(* 
| :Description: This function block represent basic TCP/IP client. 
| Use MR_Init to connect to the server. 
| To send data to server use MR_AppendToSendBuffer, use FUN_StringToTcpBufferData to convert string into structure of bytes.
| If the lenght of LastRecivedMessage is bigger than 0 then you recived message from server, use FUN_TcpBufferDataToString to copy it to string message.
| To close the connection use MR_Abort.
*)
FUNCTION_BLOCK FB_TcpClient EXTENDS FB_TcpDevice
VAR		
	(* Function blocks *)
	fbSocketConnect : FB_SocketConnect;		(* FB used to connect the client to remote server *)
END_VAR
(*
Version history:

+-------------+------------+----------------+----------+-------------------------------------------------------------------------------------+
|Date         | Version    | created under  | Author   | Remark                                                                              |
+=============+============+================+==========+=====================================================================================+
|2022-01      | 1.0.0.0    | V3.1.4024.22   | ADBO     | Function block created                                                              |
+-------------+------------+----------------+----------+-------------------------------------------------------------------------------------+
|2022-02      | 1.1.0.0    | V3.1.4024.22   | ADBO     | - Added fixes to init failure reset (MS_Aborting)                                   |
|             |            |                |          | - Changed aproach in executing all FB's ( Deleted checking error before executing ) |
+-------------+------------+----------------+----------+-------------------------------------------------------------------------------------+

*)

SUPER^();

METHOD PROTECTED MS_Aborting
IF bInitFailed THEN
	fbSocketConnect( bExecute := FALSE);
	eTcpDeviceState := TCPIP_DEVICE_UNINITIALIZED;
	
ELSE
	stSocketToClose := stHSocket;
	SUPER^.MS_Aborting();
	
END_IF
END_METHOD

(* TCP/IP client is preparing to work *)
METHOD PROTECTED MS_Initializing
SUPER^.MS_Initializing();

(* Create connection socket to remote host *)
fbSocketConnect(	sSrvNetId	:= sAmsNetID,
					sRemoteHost := sHost,
					nRemotePort := iPort,
					bExecute 	:= TRUE,
					tTimeout	:= tTimeout,
					hSocket		=> stHSocket);
						
(* Socket created *)
IF NOT fbSocketConnect.bBusy AND NOT fbSocketConnect.bError THEN
	fbSocketConnect( bExecute := FALSE);
	eTcpDeviceState := TCPIP_DEVICE_READY_INITIALIZED;
	
(*Error occured while creating client socket *)
ELSIF fbSocketConnect.bError THEN
	bError := TRUE;
	iErrorID := fbSocketConnect.nErrId;
	fbAlarmCreatingClient.ipArguments.Clear().AddUDInt(iErrorID);	
	fbAlarmCreatingClient.Raise(0);
		
END_IF
END_METHOD

END_FUNCTION_BLOCK

(* stored: Version 1.1.0.1, ProductVersion 3.1.4024.9
   POU FB_TcpClient: Id {50810698-82d6-42eb-b406-1fc109fbf32e}, SpecialFunc None
   Folder StateMachine: Id {dde683d4-89d4-443b-82d3-86337c59f2e7}
   Method MS_Aborting: Id {693ead63-edb0-47c7-899d-d767843794b9}
   Method MS_Initializing: Id {51afae26-1363-48f6-957b-4a5b997ef07d} *)
